{attribute 'GeneratedUsingTerminal: IODEVICETYPE_ETHERCATPROT'}
{attribute addProperty BoxType "IODEVICETYPE_ETHERCATPROT"}
{attribute addProperty Id "Beckhoff_EPP1xxxBeckhoff_EPP1xxx_3250354D762Beckhoff_EPP2xxxBeckhoff_EPP2xxx_8ED37E642100Beckhoff_EPP3xxxBeckhoff_EPP3xxx_37FEE8A01480Beckhoff_EPP4xxxBeckhoff_EPP4xxx_F05B7AA2222Beckhoff_EPP5xxxBeckhoff_EPP5xxx_CECB1C9F304Beckhoff_EPP6xxxBeckhoff_EPP6xxx_4A538F0B672Beckhoff_EPP7xxxBeckhoff_EPP7xxx_26C654D6550Beckhoff_EPP9xxxBeckhoff_EPP9xxx_3F2579D7102SyncUnitsSyncUnits_99E584AF18InputsInputs_25A0042B160OutputsOutputs_2397A10E106InfoDataInfoData_E68C61CD28"}
{attribute addProperty CRC "2593086843"}
{attribute addProperty Size "6504"}
TYPE EtherCAT_Master_EPPxxxx_9A8F5D7B EXTENDS EtcMasterBase_62654B43 :
STRUCT
	{attribute addProperty Name "Beckhoff EPP1xxx"}
	{attribute addProperty PreviousPort "EtherCAT_Master_EPPxxxx : Master"}
	Beckhoff_EPP1xxx : Beckhoff_EPP1xxx_3250354D;
	{attribute addProperty Name "Beckhoff EPP2xxx"}
	{attribute addProperty PreviousPort "Beckhoff EPP1xxx : C"}
	Beckhoff_EPP2xxx : Beckhoff_EPP2xxx_8ED37E64;
	{attribute addProperty Name "Beckhoff EPP3xxx"}
	{attribute addProperty PreviousPort "Beckhoff EPP2xxx : C"}
	Beckhoff_EPP3xxx : Beckhoff_EPP3xxx_37FEE8A0;
	{attribute addProperty Name "Beckhoff EPP4xxx"}
	{attribute addProperty PreviousPort "Beckhoff EPP3xxx : C"}
	Beckhoff_EPP4xxx : Beckhoff_EPP4xxx_F05B7AA2;
	{attribute addProperty Name "Beckhoff EPP5xxx"}
	{attribute addProperty PreviousPort "Beckhoff EPP4xxx : C"}
	Beckhoff_EPP5xxx : Beckhoff_EPP5xxx_CECB1C9F;
	{attribute addProperty Name "Beckhoff EPP6xxx"}
	{attribute addProperty PreviousPort "Beckhoff EPP5xxx : C"}
	Beckhoff_EPP6xxx : Beckhoff_EPP6xxx_4A538F0B;
	{attribute addProperty Name "Beckhoff EPP7xxx"}
	{attribute addProperty PreviousPort "Beckhoff EPP6xxx : C"}
	Beckhoff_EPP7xxx : Beckhoff_EPP7xxx_26C654D6;
	{attribute addProperty Name "Beckhoff EPP9xxx"}
	{attribute addProperty PreviousPort "Beckhoff EPP7xxx : C"}
	Beckhoff_EPP9xxx : Beckhoff_EPP9xxx_3F2579D7;
	{attribute addProperty Name "SyncUnits"}
	SyncUnits : SyncUnits_99E584AF;
	{attribute addProperty Name "Inputs"}
	Inputs : Inputs_25A0042B;
	{attribute addProperty Name "Outputs"}
	Outputs : Outputs_2397A10E;
	{attribute addProperty Name "InfoData"}
	InfoData : InfoData_E68C61CD;
END_STRUCT
END_TYPE

(* stored: Version 1.2.0.0, ProductVersion 3.1.4024.9
   DUT EtherCAT_Master_EPPxxxx_9A8F5D7B: Id {e79751d4-80ba-447a-bf37-87ca9a0900f3} *)
